(* This Function Block evaluates the ILK condition of the Turbo Gate valve *)
(* The logic Protects the Turbo pump from inlet pressure above the SP*)

FUNCTION F_TurboGateValve_ILK_1 : BOOL (* function return TRUE when ILK is OK*)
VAR_INPUT
	i_Turbo : ST_PTM; // Turbo Pump
	i_stISG : ST_VG; //Gauge measuring inlet Pressure e.g Pirani
END_VAR
VAR
END_VAR

(* This Function Block evaluates the ILK condition of the Turbo Gate valve *)
(* The logic Protects the Turbo pump from inlet pressure above the SP*)
F_TurboGateValve_ILK := (NOT (i_Turbo.eState = pumpSTOPPED) AND NOT (i_Turbo.eState = pumpFAULT))
						AND (i_stISG.xPRESS_OK AND i_stISG.rPRESS < i_Turbo.rInletPressureSP);

END_FUNCTION

(* stored: Version 1.1.0.1, ProductVersion 3.1.4022.18
   POU F_TurboGateValve_ILK_1: Id {4de2a450-fc41-4873-a7d2-9cd8db4a93ca}, SpecialFunc None *)
